(* PLC project marvel, Institute of Astronomy Onto 0.0.1 *)
(* stored: creationDateTime 2025-01-01T00:00:00.0, modificationDateTime 2025-01-01T00:00:00.0 *)

TYPE MarvelParts : STRUCT
  {attribute 'TcHmiSymbol.Show'}
  u1 : Unit;  (* Unit 1 *)
  {attribute 'TcHmiSymbol.Show'}
  u2 : Unit;  (* Unit 2 *)
  {attribute 'TcHmiSymbol.Show'}
  u3 : Unit;  (* Unit 3 *)
  {attribute 'TcHmiSymbol.Show'}
  u4 : Unit;  (* Unit 4 *)
  {attribute 'TcHmiSymbol.Show'}
  STCU : STCU;  (* The STCU *)
  {attribute 'TcHmiSymbol.Show'}
  services : Services;  (* Services *)
  {attribute 'TcHmiSymbol.Show'}
  sequencer : Sequencer;  (* The main sequencer of Marvel *)
  {attribute 'TcHmiSymbol.Show'}
  configManager : ConfigManager;  (* The config manager (to load/save/activate configuration data) *)
END_STRUCT;
END_TYPE

TYPE MarvelProcesses : STRUCT
  {attribute 'TcHmiSymbol.Show'}
  initialize : Process;  (* Start initializing the whole MTCS *)
  {attribute 'TcHmiSymbol.Show'}
  lock : Process;  (* Lock the whole MTCS *)
  {attribute 'TcHmiSymbol.Show'}
  unlock : Process;  (* Unlock the whole MTCS *)
  {attribute 'TcHmiSymbol.Show'}
  changeOperator : ChangeOperatorStateProcess;  (* Change the operator (e.g. OBSERVER, TECH, ...) *)
  {attribute 'TcHmiSymbol.Show'}
  verifyPassword : ChangeOperatorStateProcess;  (* Only verify the operator password *)
  {attribute 'TcHmiSymbol.Show'}
  wakeUp : Process;  (* Wake up the whole Marvel TCS *)
  {attribute 'TcHmiSymbol.Show'}
  goToSleep : Process;  (* Let the whole Marvel TCS go to sleep *)
  {attribute 'TcHmiSymbol.Show'}
  emergencyClose : Process;  (* Close all domes asap *)
  {attribute 'TcHmiSymbol.Show'}
  point : MarvelPointProcess;  (* Point multiple units at once *)
  {attribute 'TcHmiSymbol.Show'}
  openDomes : MarvelMultiUnitProcess;  (* Open the dome of multiple units at once *)
  {attribute 'TcHmiSymbol.Show'}
  closeDomes : MarvelMultiUnitProcess;  (* Close the dome of multiple units at once *)
  {attribute 'TcHmiSymbol.Show'}
  stopDomes : MarvelMultiUnitProcess;  (* Stop the dome of multiple units at once *)
END_STRUCT;
END_TYPE

TYPE MarvelStatuses : STRUCT
  {attribute 'OPC.UA.DA' := '1'}
  {attribute 'OPC.UA.DA.Access' := '1'}
  {attribute 'TcHmiSymbol.Show'}
  init : InitializationStatus;
  {attribute 'OPC.UA.DA' := '1'}
  {attribute 'OPC.UA.DA.Access' := '1'}
  {attribute 'TcHmiSymbol.Show'}
  health : HealthStatus;
  {attribute 'OPC.UA.DA' := '1'}
  {attribute 'OPC.UA.DA.Access' := '1'}
  {attribute 'TcHmiSymbol.Show'}
  busy : BusyStatus;
  {attribute 'OPC.UA.DA' := '1'}
  {attribute 'OPC.UA.DA.Access' := '1'}
  {attribute 'TcHmiSymbol.Show'}
  operator : OperatorStatus;
  {attribute 'OPC.UA.DA' := '1'}
  {attribute 'OPC.UA.DA.Access' := '1'}
  {attribute 'TcHmiSymbol.Show'}
  passwordHealth : HealthStatus;
  {attribute 'OPC.UA.DA' := '1'}
  {attribute 'OPC.UA.DA.Access' := '1'}
  {attribute 'TcHmiSymbol.Show'}
  activity : ActivityStatus;
  {attribute 'OPC.UA.DA' := '1'}
  {attribute 'OPC.UA.DA.Access' := '1'}
  {attribute 'TcHmiSymbol.Show'}
  shuttersHealth : HealthStatus;
  {attribute 'OPC.UA.DA' := '1'}
  {attribute 'OPC.UA.DA.Access' := '1'}
  {attribute 'TcHmiSymbol.Show'}
  shuttersBusy : BusyStatus;
  {attribute 'OPC.UA.DA' := '1'}
  {attribute 'OPC.UA.DA.Access' := '1'}
  {attribute 'TcHmiSymbol.Show'}
  shuttersAperture : ApertureStatus;
END_STRUCT;
END_TYPE

TYPE MarvelConfig : STRUCT
  {attribute 'TcHmiSymbol.Show'}
  endOfNightId : STRING(30);  (* ID of the EndOfNight procedure0 *)
END_STRUCT;
END_TYPE

TYPE MarvelPointProcessArgs : STRUCT
  {attribute 'TcHmiSymbol.Show'}
  alpha : LREAL;  (* Right ascention, in hours *)
  {attribute 'TcHmiSymbol.Show'}
  delta : LREAL;  (* Declination, in degrees *)
  {attribute 'TcHmiSymbol.Show'}
  u1 : BOOL;  (* True to point Unit 1 *)
  {attribute 'TcHmiSymbol.Show'}
  u2 : BOOL;  (* True to point Unit 2 *)
  {attribute 'TcHmiSymbol.Show'}
  u3 : BOOL;  (* True to point Unit 3 *)
  {attribute 'TcHmiSymbol.Show'}
  u4 : BOOL;  (* True to point Unit 4 *)
END_STRUCT;
END_TYPE

TYPE MarvelMultiUnitProcessArgs : STRUCT
  {attribute 'TcHmiSymbol.Show'}
  u1 : BOOL;  (* True to use Unit 1 *)
  {attribute 'TcHmiSymbol.Show'}
  u2 : BOOL;  (* True to use Unit 2 *)
  {attribute 'TcHmiSymbol.Show'}
  u3 : BOOL;  (* True to use Unit 3 *)
  {attribute 'TcHmiSymbol.Show'}
  u4 : BOOL;  (* True to use Unit 4 *)
END_STRUCT;
END_TYPE

TYPE M_SM_Marvel : STRUCT
  {attribute 'OPC.UA.DA' := '1'}
  {attribute 'OPC.UA.DA.Access' := '3'}
  {attribute 'TcHmiSymbol.Show'}
  editableConfig : MarvelConfig;
  {attribute 'OPC.UA.DA' := '1'}
  {attribute 'OPC.UA.DA.Access' := '1'}
  {attribute 'TcHmiSymbol.Show'}
  actualStatus : STRING;
  {attribute 'OPC.UA.DA' := '1'}
  {attribute 'OPC.UA.DA.Access' := '1'}
  {attribute 'TcHmiSymbol.Show'}
  noOfFailedOperatorChanges : UINT;
  {attribute 'OPC.UA.DA' := '1'}
  {attribute 'OPC.UA.DA.Access' := '1'}
  {attribute 'TcHmiSymbol.Show'}
  shuttersStatus : STRING;
  {attribute 'OPC.UA.DA' := '1'}
  {attribute 'OPC.UA.DA.Access' := '1'}
  {attribute 'TcHmiSymbol.Show'}
  config : MarvelConfig;
  {attribute 'OPC.UA.DA' := '1'}
  {attribute 'TcHmiSymbol.Show'}
  stat : MarvelStatuses;
  {attribute 'OPC.UA.DA' := '1'}
  {attribute 'TcHmiSymbol.Show'}
  parts : M_SM_MarvelParts;
  {attribute 'OPC.UA.DA' := '1'}
  {attribute 'TcHmiSymbol.Show'}
  proc : M_SM_MarvelProcesses;
END_STRUCT;
END_TYPE

TYPE M_MarvelPointProcess : STRUCT
  {attribute 'OPC.UA.DA' := '1'}
  {attribute 'OPC.UA.DA.Access' := '3'}
  {attribute 'TcHmiSymbol.Show'}
  set : MarvelPointProcessArgs;
END_STRUCT;
END_TYPE

TYPE M_MarvelMultiUnitProcess : STRUCT
  {attribute 'OPC.UA.DA' := '1'}
  {attribute 'OPC.UA.DA.Access' := '3'}
  {attribute 'TcHmiSymbol.Show'}
  set : MarvelMultiUnitProcessArgs;
END_STRUCT;
END_TYPE

TYPE M_SM_MarvelParts : STRUCT
  {attribute 'TcHmiSymbol.Show'}
  u1 : M_Unit;
  {attribute 'TcHmiSymbol.Show'}
  u2 : M_Unit;
  {attribute 'TcHmiSymbol.Show'}
  u3 : M_Unit;
  {attribute 'TcHmiSymbol.Show'}
  u4 : M_Unit;
  {attribute 'TcHmiSymbol.Show'}
  STCU : M_STCU;
  {attribute 'TcHmiSymbol.Show'}
  services : M_Services;
  {attribute 'TcHmiSymbol.Show'}
  sequencer : M_Sequencer;
  {attribute 'TcHmiSymbol.Show'}
  configManager : M_ConfigManager;
END_STRUCT;
END_TYPE

TYPE M_SM_MarvelProcesses : STRUCT
  {attribute 'TcHmiSymbol.Show'}
  initialize : M_Process;
  {attribute 'TcHmiSymbol.Show'}
  lock : M_Process;
  {attribute 'TcHmiSymbol.Show'}
  unlock : M_Process;
  {attribute 'TcHmiSymbol.Show'}
  changeOperator : M_ChangeOperatorStateProcess;
  {attribute 'TcHmiSymbol.Show'}
  verifyPassword : M_ChangeOperatorStateProcess;
  {attribute 'TcHmiSymbol.Show'}
  wakeUp : M_Process;
  {attribute 'TcHmiSymbol.Show'}
  goToSleep : M_Process;
  {attribute 'TcHmiSymbol.Show'}
  emergencyClose : M_Process;
  {attribute 'TcHmiSymbol.Show'}
  point : M_MarvelPointProcess;
  {attribute 'TcHmiSymbol.Show'}
  openDomes : M_MarvelMultiUnitProcess;
  {attribute 'TcHmiSymbol.Show'}
  closeDomes : M_MarvelMultiUnitProcess;
  {attribute 'TcHmiSymbol.Show'}
  stopDomes : M_MarvelMultiUnitProcess;
END_STRUCT;
END_TYPE

FUNCTION_BLOCK SM_Marvel
  VAR_INPUT
    {attribute 'OPC.UA.DA' := '1'}
    {attribute 'OPC.UA.DA.Access' := '3'}
    editableConfig : MarvelConfig;  (* Editable configuration *)
  END_VAR
  VAR_OUTPUT
    {attribute 'OPC.UA.DA' := '1'}
    {attribute 'OPC.UA.DA.Access' := '1'}
    actualStatus : STRING(50);  (* Current status description *)
    {attribute 'OPC.UA.DA' := '1'}
    {attribute 'OPC.UA.DA.Access' := '1'}
    noOfFailedOperatorChanges : UINT;  (* How many times has a wrong password been entered? *)
    {attribute 'OPC.UA.DA' := '1'}
    {attribute 'OPC.UA.DA.Access' := '1'}
    shuttersStatus : STRING(16);  (* Summary of the domes open/closed state *)
    {attribute 'OPC.UA.DA' := '1'}
    {attribute 'OPC.UA.DA.Access' := '1'}
    config : MarvelConfig;  (* Active configuration *)
    {attribute 'OPC.UA.DA' := '1'}
    stat : MarvelStatuses;  (* Statuses of the state machine *)
    {attribute 'OPC.UA.DA' := '1'}
    parts : MarvelParts;  (* Parts of the state machine *)
    {attribute 'OPC.UA.DA' := '1'}
    proc : MarvelProcesses;  (* Processes of the state machine *)
  END_VAR

            parts.u1(
    number := 1,
    operator_ref := stat.operator,
    activity_ref := stat.activity,
    services_ref := parts.services);
parts.u2(
    number := 2,
    operator_ref := stat.operator,
    activity_ref := stat.activity,
    services_ref := parts.services);
parts.u3(
    number := 3,
    operator_ref := stat.operator,
    activity_ref := stat.activity,
    services_ref := parts.services);
parts.u4(
    number := 4,
    operator_ref := stat.operator,
    activity_ref := stat.activity,
    services_ref := parts.services);
parts.STCU(
    activity_ref := stat.activity,
    services_ref := parts.services);
parts.services( operator_ref := stat.operator );
parts.sequencer( isEnabled := TRUE );
parts.configManager( isEnabled := stat.operator = OperatorStatus.tech );
stat.health := F_HealthStatus(
    superState := NOT(stat.init = InitializationStatus.shutdown),
    isGood := (NOT(stat.init = InitializationStatus.initializingFailed)) AND (((parts.u1.stat.health = HealthStatus.good) OR (parts.u1.stat.health = HealthStatus.warning)) AND (((parts.u2.stat.health = HealthStatus.good) OR (parts.u2.stat.health = HealthStatus.warning)) AND (((parts.u3.stat.health = HealthStatus.good) OR (parts.u3.stat.health = HealthStatus.warning)) AND (((parts.u4.stat.health = HealthStatus.good) OR (parts.u4.stat.health = HealthStatus.warning)) AND (((parts.services.stat.health = HealthStatus.good) OR (parts.services.stat.health = HealthStatus.warning)) AND (((parts.configManager.stat.health = HealthStatus.good) OR (parts.configManager.stat.health = HealthStatus.warning)) AND ((parts.sequencer.stat.health = HealthStatus.good) OR (parts.sequencer.stat.health = HealthStatus.warning)))))))),
    hasWarning := (parts.u1.stat.health = HealthStatus.warning) OR ((parts.u2.stat.health = HealthStatus.warning) OR ((parts.u3.stat.health = HealthStatus.warning) OR ((parts.u4.stat.health = HealthStatus.warning) OR ((parts.services.stat.health = HealthStatus.warning) OR ((parts.configManager.stat.health = HealthStatus.warning) OR (parts.sequencer.stat.health = HealthStatus.warning)))))));
stat.busy := F_BusyStatus(
    superState := NOT(stat.init = InitializationStatus.shutdown),
    isBusy := (parts.u1.stat.busy = BusyStatus.busy) OR ((parts.u2.stat.busy = BusyStatus.busy) OR ((parts.u3.stat.busy = BusyStatus.busy) OR ((parts.u4.stat.busy = BusyStatus.busy) OR ((parts.services.stat.busy = BusyStatus.busy) OR ((parts.configManager.stat.busy = BusyStatus.busy) OR (parts.sequencer.stat.busy = BusyStatus.busy)))))));
stat.shuttersHealth := F_HealthStatus(
    superState := NOT(stat.init = InitializationStatus.shutdown),
    isGood := ((parts.u1.parts.dome.parts.shutter.stat.health = HealthStatus.good) OR (parts.u1.parts.dome.parts.shutter.stat.health = HealthStatus.warning)) AND (((parts.u2.parts.dome.parts.shutter.stat.health = HealthStatus.good) OR (parts.u2.parts.dome.parts.shutter.stat.health = HealthStatus.warning)) AND (((parts.u3.parts.dome.parts.shutter.stat.health = HealthStatus.good) OR (parts.u3.parts.dome.parts.shutter.stat.health = HealthStatus.warning)) AND ((parts.u4.parts.dome.parts.shutter.stat.health = HealthStatus.good) OR (parts.u4.parts.dome.parts.shutter.stat.health = HealthStatus.warning)))),
    hasWarning := (parts.u1.parts.dome.parts.shutter.stat.health = HealthStatus.warning) OR ((parts.u2.parts.dome.parts.shutter.stat.health = HealthStatus.warning) OR ((parts.u3.parts.dome.parts.shutter.stat.health = HealthStatus.warning) OR (parts.u4.parts.dome.parts.shutter.stat.health = HealthStatus.warning))));
stat.shuttersBusy := F_BusyStatus(
    superState := NOT(stat.init = InitializationStatus.shutdown),
    isBusy := (parts.u1.parts.dome.parts.shutter.stat.busy = BusyStatus.busy) OR ((parts.u2.parts.dome.parts.shutter.stat.busy = BusyStatus.busy) OR ((parts.u3.parts.dome.parts.shutter.stat.busy = BusyStatus.busy) OR (parts.u4.parts.dome.parts.shutter.stat.busy = BusyStatus.busy))));
stat.shuttersAperture := F_ApertureStatus(
    superState := NOT(stat.init = InitializationStatus.shutdown),
    isOpen := (parts.u1.parts.dome.parts.shutter.stat.aperture = ApertureStatus.open) OR ((parts.u2.parts.dome.parts.shutter.stat.aperture = ApertureStatus.open) OR ((parts.u3.parts.dome.parts.shutter.stat.aperture = ApertureStatus.open) OR ((parts.u4.parts.dome.parts.shutter.stat.aperture = ApertureStatus.open) OR ((parts.u1.parts.dome.parts.shutter.stat.aperture = ApertureStatus.partiallyOpen) OR ((parts.u2.parts.dome.parts.shutter.stat.aperture = ApertureStatus.partiallyOpen) OR ((parts.u3.parts.dome.parts.shutter.stat.aperture = ApertureStatus.partiallyOpen) OR (parts.u4.parts.dome.parts.shutter.stat.aperture = ApertureStatus.partiallyOpen))))))),
    isClosed := (parts.u1.parts.dome.parts.shutter.stat.aperture = ApertureStatus.closed) AND ((parts.u2.parts.dome.parts.shutter.stat.aperture = ApertureStatus.closed) AND ((parts.u3.parts.dome.parts.shutter.stat.aperture = ApertureStatus.closed) AND (parts.u4.parts.dome.parts.shutter.stat.aperture = ApertureStatus.closed))));
proc.initialize( isEnabled := NOT(stat.init = InitializationStatus.initializing) );
proc.lock( isEnabled := (stat.operator = OperatorStatus.tech) AND (stat.init = InitializationStatus.initialized) );
proc.unlock( isEnabled := (stat.operator = OperatorStatus.tech) AND (stat.init = InitializationStatus.locked) );
proc.changeOperator( isEnabled := TRUE );
proc.verifyPassword( isEnabled := TRUE );
proc.wakeUp( isEnabled := TRUE );
proc.goToSleep( isEnabled := TRUE );
proc.emergencyClose( isEnabled := NOT((parts.u1.parts.dome.parts.shutter.stat.aperture = ApertureStatus.closed) AND ((parts.u1.parts.dome.parts.shutter.stat.aperture = ApertureStatus.closed) AND ((parts.u1.parts.dome.parts.shutter.stat.aperture = ApertureStatus.closed) AND (parts.u1.parts.dome.parts.shutter.stat.aperture = ApertureStatus.closed)))) );
proc.point( isEnabled := parts.u1.proc.point.isEnabled OR (parts.u2.proc.point.isEnabled OR (parts.u3.proc.point.isEnabled OR parts.u4.proc.point.isEnabled)) );
proc.openDomes( isEnabled := parts.u1.parts.dome.parts.shutter.proc.open.isEnabled OR (parts.u2.parts.dome.parts.shutter.proc.open.isEnabled OR (parts.u3.parts.dome.parts.shutter.proc.open.isEnabled OR parts.u4.parts.dome.parts.shutter.proc.open.isEnabled)) );
proc.closeDomes( isEnabled := parts.u1.parts.dome.parts.shutter.proc.close.isEnabled OR (parts.u2.parts.dome.parts.shutter.proc.close.isEnabled OR (parts.u3.parts.dome.parts.shutter.proc.close.isEnabled OR parts.u4.parts.dome.parts.shutter.proc.close.isEnabled)) );
proc.stopDomes( isEnabled := parts.u1.parts.dome.parts.shutter.proc.stop.isEnabled OR (parts.u2.parts.dome.parts.shutter.proc.stop.isEnabled OR (parts.u3.parts.dome.parts.shutter.proc.stop.isEnabled OR parts.u4.parts.dome.parts.shutter.proc.stop.isEnabled)) );

          

METHOD _copyFromModel_SM_Marvel
  VAR_IN_OUT
    {attribute 'OPC.UA.DA' := '0'}
    model : M_SM_Marvel;
  END_VAR
                  THIS^.editableConfig := model.editableConfig;
THIS^.parts.u1._copyFromModel_Unit( model := model.parts.u1 );
THIS^.parts.u2._copyFromModel_Unit( model := model.parts.u2 );
THIS^.parts.u3._copyFromModel_Unit( model := model.parts.u3 );
THIS^.parts.u4._copyFromModel_Unit( model := model.parts.u4 );
THIS^.parts.STCU._copyFromModel_STCU( model := model.parts.STCU );
THIS^.parts.services._copyFromModel_Services( model := model.parts.services );
THIS^.parts.sequencer._copyFromModel_Sequencer( model := model.parts.sequencer );
THIS^.parts.configManager._copyFromModel_ConfigManager( model := model.parts.configManager );
THIS^.proc.initialize._copyFromModel_Process( model := model.proc.initialize );
THIS^.proc.lock._copyFromModel_Process( model := model.proc.lock );
THIS^.proc.unlock._copyFromModel_Process( model := model.proc.unlock );
THIS^.proc.changeOperator._copyFromModel_ChangeOperatorStateProcess( model := model.proc.changeOperator );
THIS^.proc.verifyPassword._copyFromModel_ChangeOperatorStateProcess( model := model.proc.verifyPassword );
THIS^.proc.wakeUp._copyFromModel_Process( model := model.proc.wakeUp );
THIS^.proc.goToSleep._copyFromModel_Process( model := model.proc.goToSleep );
THIS^.proc.emergencyClose._copyFromModel_Process( model := model.proc.emergencyClose );
THIS^.proc.point._copyFromModel_MarvelPointProcess( model := model.proc.point );
THIS^.proc.openDomes._copyFromModel_MarvelMultiUnitProcess( model := model.proc.openDomes );
THIS^.proc.closeDomes._copyFromModel_MarvelMultiUnitProcess( model := model.proc.closeDomes );
THIS^.proc.stopDomes._copyFromModel_MarvelMultiUnitProcess( model := model.proc.stopDomes );

                
END_METHOD

METHOD _copyToModel_SM_Marvel
  VAR_IN_OUT
    {attribute 'OPC.UA.DA' := '0'}
    model : M_SM_Marvel;
  END_VAR
                  model.editableConfig := THIS^.editableConfig;
model.actualStatus := THIS^.actualStatus;
model.noOfFailedOperatorChanges := THIS^.noOfFailedOperatorChanges;
model.shuttersStatus := THIS^.shuttersStatus;
model.config := THIS^.config;
model.stat := THIS^.stat;
THIS^.parts.u1._copyToModel_Unit( model := model.parts.u1 );
THIS^.parts.u2._copyToModel_Unit( model := model.parts.u2 );
THIS^.parts.u3._copyToModel_Unit( model := model.parts.u3 );
THIS^.parts.u4._copyToModel_Unit( model := model.parts.u4 );
THIS^.parts.STCU._copyToModel_STCU( model := model.parts.STCU );
THIS^.parts.services._copyToModel_Services( model := model.parts.services );
THIS^.parts.sequencer._copyToModel_Sequencer( model := model.parts.sequencer );
THIS^.parts.configManager._copyToModel_ConfigManager( model := model.parts.configManager );
THIS^.proc.initialize._copyToModel_Process( model := model.proc.initialize );
THIS^.proc.lock._copyToModel_Process( model := model.proc.lock );
THIS^.proc.unlock._copyToModel_Process( model := model.proc.unlock );
THIS^.proc.changeOperator._copyToModel_ChangeOperatorStateProcess( model := model.proc.changeOperator );
THIS^.proc.verifyPassword._copyToModel_ChangeOperatorStateProcess( model := model.proc.verifyPassword );
THIS^.proc.wakeUp._copyToModel_Process( model := model.proc.wakeUp );
THIS^.proc.goToSleep._copyToModel_Process( model := model.proc.goToSleep );
THIS^.proc.emergencyClose._copyToModel_Process( model := model.proc.emergencyClose );
THIS^.proc.point._copyToModel_MarvelPointProcess( model := model.proc.point );
THIS^.proc.openDomes._copyToModel_MarvelMultiUnitProcess( model := model.proc.openDomes );
THIS^.proc.closeDomes._copyToModel_MarvelMultiUnitProcess( model := model.proc.closeDomes );
THIS^.proc.stopDomes._copyToModel_MarvelMultiUnitProcess( model := model.proc.stopDomes );

                
END_METHOD
END_FUNCTION_BLOCK

FUNCTION_BLOCK MarvelPointProcess EXTENDS BaseProcess
  VAR_INPUT
    {attribute 'OPC.UA.DA' := '1'}
    {attribute 'OPC.UA.DA.Access' := '3'}
    {attribute 'TcHmiSymbol.Show'}
    set : MarvelPointProcessArgs;  (* Arguments to be set, before writing do_request TRUE *)
  END_VAR
  VAR_OUTPUT
    {attribute 'OPC.UA.DA' := '0'}
    get : MarvelPointProcessArgs;  (* Arguments in use by the process, if do_request was accepted *)
  END_VAR

            IF do_request THEN
    do_request_result := request(
    alpha := set.alpha,
    delta := set.delta,
    u1 := set.u1,
    u2 := set.u2,
    u3 := set.u3,
    u4 := set.u4);
    do_request := FALSE;
END_IF;
SUPER^();

          

{attribute 'TcRpcEnable' := '1'}
METHOD start
  VAR_INPUT
    alpha : LREAL;  (* Right ascention, in hours *)
    delta : LREAL;  (* Declination, in degrees *)
    u1 : BOOL;  (* True to point Unit 1 *)
    u2 : BOOL;  (* True to point Unit 2 *)
    u3 : BOOL;  (* True to point Unit 3 *)
    u4 : BOOL;  (* True to point Unit 4 *)
  END_VAR
                  THIS^.get.alpha := alpha;
THIS^.get.delta := delta;
THIS^.get.u1 := u1;
THIS^.get.u2 := u2;
THIS^.get.u3 := u3;
THIS^.get.u4 := u4;
THIS^.stat.busy := BusyStatus.busy;
THIS^.stat.health := HealthStatus.good;

                
END_METHOD

{attribute 'TcRpcEnable' := '1'}
METHOD request : RequestResults
  VAR_INPUT
    alpha : LREAL;  (* Right ascention, in hours *)
    delta : LREAL;  (* Declination, in degrees *)
    u1 : BOOL;  (* True to point Unit 1 *)
    u2 : BOOL;  (* True to point Unit 2 *)
    u3 : BOOL;  (* True to point Unit 3 *)
    u4 : BOOL;  (* True to point Unit 4 *)
  END_VAR
                  IF THIS^.stat.enabled = EnabledStatus.enabled THEN
    request := RequestResults.ACCEPTED;
    THIS^.start(
        alpha := alpha,
        delta := delta,
        u1 := u1,
        u2 := u2,
        u3 := u3,
        u4 := u4);
ELSE
    request := RequestResults.REJECTED;
END_IF;

                
END_METHOD

METHOD _copyFromModel_MarvelPointProcess
  VAR_IN_OUT
    {attribute 'OPC.UA.DA' := '0'}
    model : M_MarvelPointProcess;
  END_VAR
                  THIS^.set := model.set;
SUPER^._copyFromModel_BaseProcess( model := model );

                
END_METHOD

METHOD _copyToModel_MarvelPointProcess
  VAR_IN_OUT
    {attribute 'OPC.UA.DA' := '0'}
    model : M_MarvelPointProcess;
  END_VAR
                  model.set := THIS^.set;
SUPER^._copyToModel_BaseProcess( model := model );

                
END_METHOD
END_FUNCTION_BLOCK

FUNCTION_BLOCK MarvelMultiUnitProcess EXTENDS BaseProcess
  VAR_INPUT
    {attribute 'OPC.UA.DA' := '1'}
    {attribute 'OPC.UA.DA.Access' := '3'}
    {attribute 'TcHmiSymbol.Show'}
    set : MarvelMultiUnitProcessArgs;  (* Arguments to be set, before writing do_request TRUE *)
  END_VAR
  VAR_OUTPUT
    {attribute 'OPC.UA.DA' := '0'}
    get : MarvelMultiUnitProcessArgs;  (* Arguments in use by the process, if do_request was accepted *)
  END_VAR

            IF do_request THEN
    do_request_result := request(
    u1 := set.u1,
    u2 := set.u2,
    u3 := set.u3,
    u4 := set.u4);
    do_request := FALSE;
END_IF;
SUPER^();

          

{attribute 'TcRpcEnable' := '1'}
METHOD start
  VAR_INPUT
    u1 : BOOL;  (* True to use Unit 1 *)
    u2 : BOOL;  (* True to use Unit 2 *)
    u3 : BOOL;  (* True to use Unit 3 *)
    u4 : BOOL;  (* True to use Unit 4 *)
  END_VAR
                  THIS^.get.u1 := u1;
THIS^.get.u2 := u2;
THIS^.get.u3 := u3;
THIS^.get.u4 := u4;
THIS^.stat.busy := BusyStatus.busy;
THIS^.stat.health := HealthStatus.good;

                
END_METHOD

{attribute 'TcRpcEnable' := '1'}
METHOD request : RequestResults
  VAR_INPUT
    u1 : BOOL;  (* True to use Unit 1 *)
    u2 : BOOL;  (* True to use Unit 2 *)
    u3 : BOOL;  (* True to use Unit 3 *)
    u4 : BOOL;  (* True to use Unit 4 *)
  END_VAR
                  IF THIS^.stat.enabled = EnabledStatus.enabled THEN
    request := RequestResults.ACCEPTED;
    THIS^.start(
        u1 := u1,
        u2 := u2,
        u3 := u3,
        u4 := u4);
ELSE
    request := RequestResults.REJECTED;
END_IF;

                
END_METHOD

METHOD _copyFromModel_MarvelMultiUnitProcess
  VAR_IN_OUT
    {attribute 'OPC.UA.DA' := '0'}
    model : M_MarvelMultiUnitProcess;
  END_VAR
                  THIS^.set := model.set;
SUPER^._copyFromModel_BaseProcess( model := model );

                
END_METHOD

METHOD _copyToModel_MarvelMultiUnitProcess
  VAR_IN_OUT
    {attribute 'OPC.UA.DA' := '0'}
    model : M_MarvelMultiUnitProcess;
  END_VAR
                  model.set := THIS^.set;
SUPER^._copyToModel_BaseProcess( model := model );

                
END_METHOD
END_FUNCTION_BLOCK
